PROGRAM MAIN
VAR
	fbConveyer : FB_Conveyer;
	fbMachineController : FB_MachineController(_iConveyer := fbConveyer);
END_VAR


fbMachineController();

END_PROGRAM

(* stored: Version 1.1.0.1, ProductVersion 3.1.4024.16
   POU MAIN: Id {8da3d096-1754-40ee-b80d-caff5cf9410f}, SpecialFunc None *)
